FUNCTION_BLOCK FB_PFEIFFER_PTM
VAR_IN_OUT
	iq_stPTM : ST_PTM;
END_VAR
VAR_INPUT
END_VAR
VAR_OUTPUT
END_VAR
VAR
END_VAR

(* Basic pump supervisory section *)
IF iq_stPTM.xExtRunOk AND NOT (iq_stPTM.xFault OR iq_stPTM.xTempFault) THEN
	iq_stPTM.q_RunDO:=iq_stPTM.i_xRunSW;
ELSE
	iq_stPTM.i_xRunSW:=0;
	iq_stPTM.q_RunDO:=FALSE;
END_IF

END_FUNCTION_BLOCK

(* stored: Version 1.1.0.1, ProductVersion 3.1.0.26
   POU FB_PFEIFFER_PTM: Id {f61aaad0-85b4-4244-b8a7-58d7d76a340e} *)
